PROGRAM main
VAR
	ESTOP AT %IX0.0 : bool;
	STOP AT %IX0.1 : bool;
	START AT %IX0.2 : bool;
	RUNNING AT %QX0.0 : bool;
	STOPPED AT %QX0.1 : bool;
	FAULT AT %QX0.2 : bool;
	FSM0 : FSM;
	START_CMD AT %QX0.3 : bool;
	STOP_CMD AT %QX0.4 : bool;
	ESTOP_CMD AT %QX0.5 : bool;
END_VAR

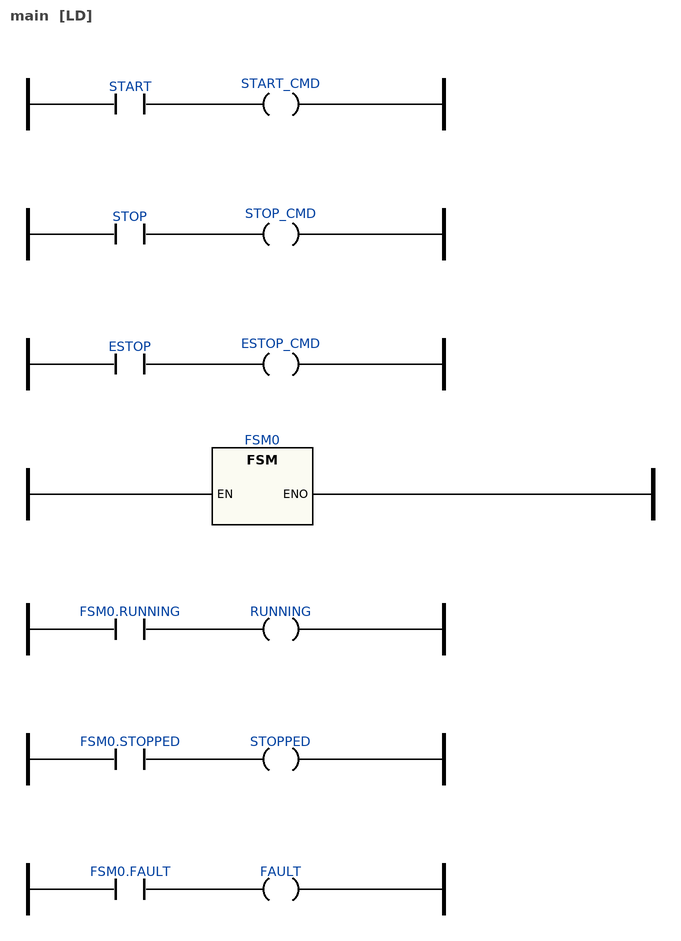
(* LD diagram, written out as Structured Text *)
START_CMD := START;
STOP_CMD := STOP;
ESTOP_CMD := ESTOP;
RUNNING := FSM0.RUNNING;
STOPPED := FSM0.STOPPED;
FAULT := FSM0.FAULT;
FSM0();
END_PROGRAM
